(* IEC 61131-3 sources: Std_PalletMover/Class/I_PiviotWheel, 1 file *)

(* ---- I_PiviotWheel.st ---- *)
(*!
<Class
	Name               = "I_PiviotWheel"
	Revision           = "0.0"
	RealtimeTask       = "false"
	CyclicTask         = "false"
	BackgroundTask     = "false"
	Sigmatek           = "false"
	OSInterface        = "false"
	HighPriority       = "false"
	Automatic          = "false"
	UpdateMode         = "Prescan"
	SharedCommandTable = "true"
	Objectsize         = "(720,120)">
	<Channels>
		<Server Name="ClassSvr" Visualized="false" Initialize="false" WriteProtected="true" Retentive="false"/>
		<Client Name="ToPiviotWheel1" Required="true" Internal="false"/>
	</Channels>
</Class>
*)
I_PiviotWheel : CLASS
  //Servers:
	ClassSvr 	: SvrChCmd_DINT;
  //Clients:
	ToPiviotWheel1 	: CltChCmd_PerPiviotWeel;
  //Variables:
  //Functions:
  //Tables:
	FUNCTION @STD
		VAR_OUTPUT
			ret_code	: CONFSTATES;
		END_VAR;
	FUNCTION GLOBAL TAB @CT_;
END_CLASS;

#pragma usingLtd PerPiviotWeel
